INTERFACE I_OutputPorts

METHOD PUBLIC Accept
VAR_INPUT
	Visitor : I_OutputPortVisitor;
END_VAR
END_METHOD

METHOD PUBLIC AddDataAsOutputPort : I_OutputPort
VAR_INPUT
	Name : T_MAXSTRING;
	Data : I_Datatype;
END_VAR
END_METHOD

METHOD AddOutputPort
VAR_INPUT
	OutputPort : I_OutputPort;
END_VAR
END_METHOD

METHOD PUBLIC TryGetOutputPortByName : BOOL
VAR_INPUT
	Name : T_MAXSTRING;
	Destination : REFERENCE TO I_OutputPort;
END_VAR
END_METHOD

END_INTERFACE

(* stored: Version 1.1.0.1, ProductVersion 3.1.4024.12
   Itf I_OutputPorts: Id {f3465273-5ac8-459b-a9cd-526bbcff246c}
   Method Accept: Id {c26dc5d0-54bb-4438-91f2-063c3970eb33}
   Method AddDataAsOutputPort: Id {f220ca25-cf69-4143-bc55-d9bc474176ae}
   Method AddOutputPort: Id {ccc39ff5-e25c-0f20-3efe-f937f75d1bdc}
   Method TryGetOutputPortByName: Id {a3a67671-970b-01d6-2705-151b345eba16} *)
